ABB RAPID module: MODULE Module1.mod

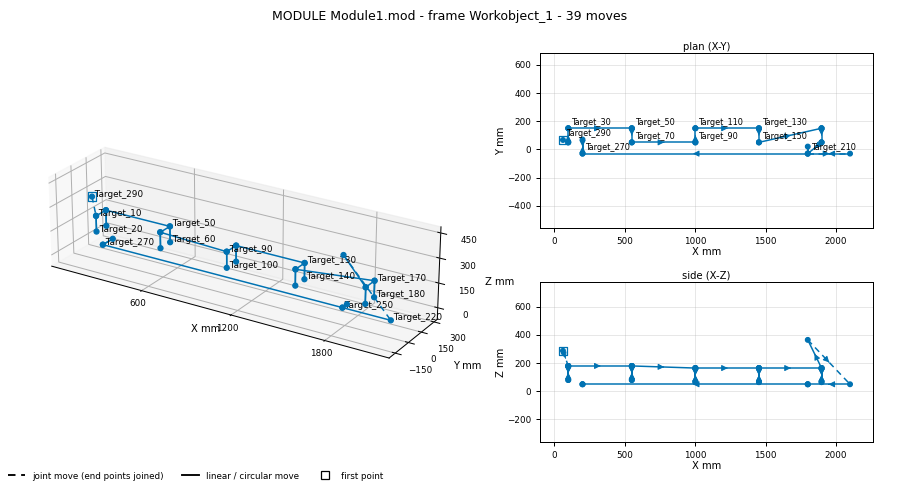
[picture p0: tool path of MODULE Module1.mod in frame Workobject_1, 39 of 39 moves have a stored position in this frame; points joined in program order, loops and branches not executed]
MODULE Module1
    CONST robtarget Target_10:=[[100,50,180],[0,0,1,0],[0,0,0,0],[0,9E+09,9E+09,9E+09,9E+09,9E+09]];
    CONST robtarget Target_20:=[[100,50,80],[0,0,1,0],[0,0,0,0],[0,9E+09,9E+09,9E+09,9E+09,9E+09]];
    CONST robtarget Target_40:=[[100,150,80],[0,0,1,0],[0,0,0,0],[0,9E+09,9E+09,9E+09,9E+09,9E+09]];
    CONST robtarget Target_30:=[[100,150,180],[0,0,1,0],[0,0,0,0],[0,9E+09,9E+09,9E+09,9E+09,9E+09]];
    CONST robtarget Target_50:=[[551.105673906,149.999980134,179.999981847],[0.000000002,0,1,0.000000008],[0,-1,0,0],[451.105651106,9E+09,9E+09,9E+09,9E+09,9E+09]];
    CONST robtarget Target_60:=[[551.105674306,149.999981734,79.999981847],[0.000000002,0,1,0.000000008],[0,-1,0,0],[451.105651106,9E+09,9E+09,9E+09,9E+09,9E+09]];
    CONST robtarget Target_70:=[[551.106,50,180],[0,0,1,0],[0,0,0,0],[451.105651106,9E+09,9E+09,9E+09,9E+09,9E+09]];
    CONST robtarget Target_80:=[[551.106,50,80],[0,0,1,0],[0,0,0,0],[451.105651106,9E+09,9E+09,9E+09,9E+09,9E+09]];
    CONST robtarget Target_90:=[[1002.211,50,165],[0,0,1,0],[0,0,0,0],[902.211302211,9E+09,9E+09,9E+09,9E+09,9E+09]];
    CONST robtarget Target_100:=[[1002.211,50,65],[0,0,1,0],[0,0,0,0],[902.211302211,9E+09,9E+09,9E+09,9E+09,9E+09]];
    CONST robtarget Target_120:=[[1002.211271152,150.000028538,64.999995901],[-0.000000004,0,1,-0.000000021],[0,-1,0,0],[902.211302211,9E+09,9E+09,9E+09,9E+09,9E+09]];
    CONST robtarget Target_110:=[[1002.211271952,150.000032738,164.999995901],[-0.000000004,0,1,-0.000000021],[0,-1,0,0],[902.211302211,9E+09,9E+09,9E+09,9E+09,9E+09]];
    CONST robtarget Target_130:=[[1453.316929894,150.000067521,164.999981784],[-0.000000004,0,1,-0.000000021],[0,-1,0,0],[1353.316953317,9E+09,9E+09,9E+09,9E+09,9E+09]];
    CONST robtarget Target_140:=[[1453.316929094,150.000063321,64.999981784],[-0.000000004,0,1,-0.000000021],[0,-1,0,0],[1353.316953317,9E+09,9E+09,9E+09,9E+09,9E+09]];
    CONST robtarget Target_150:=[[1453.317,50,165],[0,0,1,0],[0,0,0,0],[1353.316953317,9E+09,9E+09,9E+09,9E+09,9E+09]];
    CONST robtarget Target_160:=[[1453.317,50,65],[0,0,1,0],[0,0,0,0],[1353.316953317,9E+09,9E+09,9E+09,9E+09,9E+09]];
    CONST robtarget Target_170:=[[1897.788674366,150.000067521,164.999981784],[-0.000000004,0,1,-0.000000021],[0,-1,0,0],[1797.788697789,9E+09,9E+09,9E+09,9E+09,9E+09]];
    CONST robtarget Target_180:=[[1897.788673566,150.000063321,64.999981784],[-0.000000004,0,1,-0.000000021],[0,-1,0,0],[1797.788697789,9E+09,9E+09,9E+09,9E+09,9E+09]];
    CONST robtarget Target_190:=[[1897.789,50,165],[0,0,1,0],[0,0,0,0],[1797.788697789,9E+09,9E+09,9E+09,9E+09,9E+09]];
    CONST robtarget Target_200:=[[1897.789,50,65],[0,0,1,0],[0,0,0,0],[1797.788697789,9E+09,9E+09,9E+09,9E+09,9E+09]];
    CONST robtarget Target_210:=[[1800,-30,365],[0,0,1,0],[0,0,0,0],[1797.788697789,9E+09,9E+09,9E+09,9E+09,9E+09]];
    CONST robtarget Target_250:=[[1800,-30,50],[0.707106781,-0.707106781,0,0],[0,-1,-2,1],[1797.788697789,9E+09,9E+09,9E+09,9E+09,9E+09]];
    CONST robtarget Target_260:=[[1800,20,50],[0.707106781,-0.707106781,0,0],[0,-1,-2,1],[1797.788697789,9E+09,9E+09,9E+09,9E+09,9E+09]];
    CONST robtarget Target_220:=[[2100,-30,50],[0.707106781,-0.707106781,0,0],[0,-1,-1,1],[1797.788697789,9E+09,9E+09,9E+09,9E+09,9E+09]];
    CONST robtarget Target_270:=[[201.228536798,-29.999979352,49.999984645],[0.70710682,-0.707106743,0.000000006,-0.000000006],[0,-1,-2,1],[199.017199017,9E+09,9E+09,9E+09,9E+09,9E+09]];
    CONST robtarget Target_280:=[[201.228538495,70.000020648,49.999995534],[0.70710682,-0.707106743,0.000000006,-0.000000006],[0,-1,-2,1],[199.017199017,9E+09,9E+09,9E+09,9E+09,9E+09]];
    CONST robtarget Target_290:=[[62.460879069,66.841475712,287.462685107],[0.002224961,-0.987408951,-0.158108191,-0.00451816],[1,-1,-2,0],[199.017211795,9E+09,9E+09,9E+09,9E+09,9E+09]];

    PROC main()

        Path_10;
    ENDPROC
    PROC Path_10()
        MoveL Target_290,v100,z10,drillBit\WObj:=Workobject_1;
        MoveJ Target_10,v100,z10,drillBit\WObj:=Workobject_1;
        MoveL Target_20,v100,z10,drillBit\WObj:=Workobject_1;
        MoveL Target_10,v100,z10,drillBit\WObj:=Workobject_1;
        MoveL Target_30,v100,z10,drillBit\WObj:=Workobject_1;
        MoveL Target_40,v100,z10,drillBit\WObj:=Workobject_1;
        MoveL Target_30,v100,z10,drillBit\WObj:=Workobject_1;
        MoveL Target_50,v100,z10,drillBit\WObj:=Workobject_1;
        MoveL Target_60,v100,z10,drillBit\WObj:=Workobject_1;
        MoveL Target_50,v100,z10,drillBit\WObj:=Workobject_1;
        MoveL Target_70,v100,z10,drillBit\WObj:=Workobject_1;
        MoveL Target_80,v100,z10,drillBit\WObj:=Workobject_1;
        MoveL Target_70,v100,z10,drillBit\WObj:=Workobject_1;
        MoveL Target_90,v100,z10,drillBit\WObj:=Workobject_1;
        MoveL Target_100,v100,z10,drillBit\WObj:=Workobject_1;
        MoveL Target_90,v100,z10,drillBit\WObj:=Workobject_1;
        MoveL Target_110,v100,z10,drillBit\WObj:=Workobject_1;
        MoveL Target_120,v100,z10,drillBit\WObj:=Workobject_1;
        MoveL Target_110,v100,z10,drillBit\WObj:=Workobject_1;
        MoveL Target_130,v100,z10,drillBit\WObj:=Workobject_1;
        MoveL Target_140,v100,z10,drillBit\WObj:=Workobject_1;
        MoveL Target_130,v100,z10,drillBit\WObj:=Workobject_1;
        MoveL Target_150,v100,z10,drillBit\WObj:=Workobject_1;
        MoveL Target_160,v100,z10,drillBit\WObj:=Workobject_1;
        MoveL Target_150,v100,z10,drillBit\WObj:=Workobject_1;
        MoveL Target_170,v100,z10,drillBit\WObj:=Workobject_1;
        MoveL Target_180,v100,z10,drillBit\WObj:=Workobject_1;
        MoveL Target_170,v100,z10,drillBit\WObj:=Workobject_1;
        MoveL Target_190,v100,z10,drillBit\WObj:=Workobject_1;
        MoveL Target_200,v100,z10,drillBit\WObj:=Workobject_1;
        MoveL Target_190,v100,z10,drillBit\WObj:=Workobject_1;
        MoveL Target_210,v100,z10,drillBit\WObj:=Workobject_1;
        MoveJ Target_220,v100,z10,drillBit\WObj:=Workobject_1;
        MoveL Target_250,v100,z10,drillBit\WObj:=Workobject_1;
        MoveL Target_260,v100,z10,drillBit\WObj:=Workobject_1;
        MoveL Target_250,v100,z10,drillBit\WObj:=Workobject_1;
        MoveL Target_270,v100,z10,drillBit\WObj:=Workobject_1;
        MoveL Target_280,v100,z10,drillBit\WObj:=Workobject_1;
        MoveL Target_270,v100,z10,drillBit\WObj:=Workobject_1;
    ENDPROC
ENDMODULE
